INTERFACE ITF_Observer

METHOD Update : BOOL
VAR_INPUT
	TwinSAFEGroup : ITF_TwinSAFEGroup;
END_VAR
END_METHOD

END_INTERFACE

(* stored: Version 1.1.0.1, ProductVersion 3.1.4024.12
   Itf ITF_Observer: Id {22088183-9676-40aa-b065-41c25e0b52a7}
   Method Update: Id {3ae5d886-bbd4-4453-b259-c5a605e1466a} *)
